// TwinCAT 3 PLC project PLC_Main
// ProgramVersion: 3.1.4026.13
// CompilerDefines: VISU_USEWSTRING
// libraries:
//   Tc2_Standard, * (Beckhoff Automation GmbH)
//   Tc2_System, * (Beckhoff Automation GmbH)
//   Tc3_Module, * (Beckhoff Automation GmbH)
// project tree:
//   DUTs/ DUT_TestStruct.TcDUT, DUT_TestStruct2.TcDUT, MonitorTest.TcDUT, MonitorTestData.TcDUT, ReadTest.TcDUT, ReadTestData.TcDUT, SymbolTest.TcDUT, TestEnum.TcDUT, WriteTest.TcDUT, WriteTestData.TcDUT
//   GVLs/ AdsNet8.TcGVL, AdsNet9.TcGVL, OpcNet8.TcGVL, OpcNet9.TcGVL
//   / PlcTask.TcTTO
//   POUs/ MAIN.TcPOU, ResetWriteData.TcPOU
// real-time tasks:
//   TASK PlcTask: cycle T#10ms, priority 20, ADS port 350

CONFIGURATION PLC_Main
    RESOURCE PLC ON TwinCAT3
        TASK PlcTask(INTERVAL := T#10ms, PRIORITY := 20);
        PROGRAM MAIN WITH PlcTask : MAIN;
    END_RESOURCE
END_CONFIGURATION

// ---- DUTs/DUT_TestStruct.TcDUT
{attribute 'analysis' := '-33'}
TYPE DUT_TestStruct :
STRUCT
	BoolValue						:BOOL			:= TRUE;
	
	ByteValue						:BYTE			:= 16#FF;
	WordValue						:WORD			:= 16#FFFF;
	DWordValue						:DWORD			:= 16#FFFF_FFFF;
	LWordValue						:LWORD			:= 16#FFFF_FFFF_FFFF_FFFF;
	
	ShortValue						:SINT			:= -128;
	IntValue						:INT			:= -32768;
	DIntValue						:DINT			:= -2147483648 ;
	LongValue						:LINT			:= -9223372036854775808;

	UShortValue						:USINT			:= 255;
	UIntValue						:UINT			:= 65535;
	UDIntValue						:UDINT			:= 4294967295;
	ULongValue						:ULINT			:= 18446744073709551615;
										   
	FloatValue						:REAL			:= -3.402823E+38;
	DoubleValue						:LREAL			:= -1.79769313486231E+308;
	
	TimeValue						:TIME			:= T#1000MS;
	TimeOfDay						:TIME_OF_DAY	:= TOD#01:00;
	LTimeValue						:LTIME 			:= LTIME#1000NS;
	DateValue						:DATE			:= D#2106-02-05;
	DateAndTimeValue				:DATE_AND_TIME	:= DT#2106-02-05-06:28:15;
	
	StringValue						:STRING			:= 'Test String';
	WStringValue					:WSTRING		:= "Test WString";
	
	Nested							:DUT_TestStruct2;
	
	IntArray						:ARRAY[0..10] OF INT := [1000, 1001, 1002, 1003, 1004, 1005, 1006, 1007, 1008, 1009, 1010];
	MultiDimensionArray 			:ARRAY[0..1,0..2,0..3] OF INT := [100, 200, 300, 400, 500, 600, 700, 800, 900, 1000, 1100, 1200, 1300, 1400, 1500, 1600, 1700, 1800, 1900, 2000, 2100, 2200, 2300, 2400];
	ComplexArray					:ARRAY[0..2] OF DUT_TestStruct2;
	MultiDimensionComplexArray 		:ARRAY[0..1,0..2,0..3] OF DUT_TestStruct2;
	
	IntArray2						:ARRAY[1..11] OF INT := [1000, 1001, 1002, 1003, 1004, 1005, 1006, 1007, 1008, 1009, 1010];
	MultiDimensionArray2			:ARRAY[1..2,1..3,1..4] OF INT := [100, 200, 300, 400, 500, 600, 700, 800, 900, 1000, 1100, 1200, 1300, 1400, 1500, 1600, 1700, 1800, 1900, 2000, 2100, 2200, 2300, 2400];
	ComplexArray2					:ARRAY[1..3] OF DUT_TestStruct2;
	MultiDimensionComplexArray2		:ARRAY[1..2,1..3,1..4] OF DUT_TestStruct2;
END_STRUCT
END_TYPE

// ---- DUTs/DUT_TestStruct2.TcDUT
{attribute 'analysis' := '-33'}
TYPE DUT_TestStruct2 :
STRUCT
	ByteValue			:BYTE			:= 16#FF;
	WordValue			:WORD			:= 16#FFFF;
	DWordValue			:DWORD			:= 16#FFFF_FFFF;
	LWordValue			:LWORD			:= 16#FFFF_FFFF_FFFF_FFFF;
END_STRUCT
END_TYPE

// ---- DUTs/MonitorTest.TcDUT
{attribute 'analysis' := '-33'}
TYPE MonitorTest :
STRUCT
    MonitorBeforeConnectDoesNotMatter			: BOOL;	
    SubscriptionsWillAllTriggerOnUpdateAsync	: BOOL;
    RegisterUnregisterIO						: BOOL;
    
    RegisterUnregisterMultipleIO1				: BOOL;
    RegisterUnregisterMultipleIO2				: BOOL;
    RegisterUnregisterMultipleIO3				: BOOL;
    RegisterUnregisterMultipleIO4				: BOOL;
    RegisterUnregisterMultipleIO5				: BOOL;
    RegisterUnregisterMultipleIO6				: BOOL;
    RegisterUnregisterMultipleIO7				: BOOL;
    RegisterUnregisterMultipleIO8				: BOOL;
    
    SubscribeIOUpdatesWhenValueChanges			: BOOL;
    SubscriptionsPersistReconnects				: BOOL;
    SubscribeIOShouldTriggerOnSubscribe			: BOOL;
    
    CanSubscribeToAllPlcTypes					: MonitorTestData;
END_STRUCT
END_TYPE

// ---- DUTs/MonitorTestData.TcDUT
{attribute 'analysis' := '-33'}
TYPE MonitorTestData :
STRUCT
	BoolValue			: BOOL;
	
	ByteValue			: BYTE;
	WordValue			: WORD;
	DWordValue			: DWORD;
	LWordValue			: LWORD;
	
	SIntValue			: SINT;
	IntValue			: INT;
	DIntValue			: DINT;
	LIntValue			: LINT;
	
	USIntValue			: USINT;
	UIntValue			: UINT;
	UDIntValue			: UDINT;
	ULIntValue			: ULINT;
	
	RealValue			: REAL;
	LRealValue			: LREAL;
	
	TimeValue			: TIME;
	TimeOfDayValue		: TOD;
	LTimeValue			: LTIME;
	DateValue			: DATE;
	DateAndTimeValue	: DT;
	StringValue			: STRING;
	WStringValue		: WSTRING;
	EnumValue1			: TestEnum;
	EnumValue2			: TestEnum;
END_STRUCT
END_TYPE

// ---- DUTs/ReadTest.TcDUT
{attribute 'analysis' := '-33'}
TYPE ReadTest :
STRUCT
	ReadDynamicReadsAStructure					: DUT_TestStruct;
	ReadDynamicReadsAStructureAsync				: DUT_TestStruct;

	ReadGenericReturnsTheRequestedType			: ReadTestData;
	ReadGenericReturnsTheRequestedTypeAsync		: ReadTestData;
	
	ReadMultipleItemsInOneTransaction			: ReadTestData;
	ReadMultipleItemsInOneTransactionAsync		: ReadTestData;
	
	ReadValueReturnsTheExpectedValue			: ReadTestData;
	ReadValueReturnsTheExpectedValueAsync		: ReadTestData;
	
	WaitForValueThrowsExceptionOnTimeout		: BOOL;
	WaitForValueThrowsExceptionOnTimeoutAsync	: BOOL;
	
	WaitsForValueToChange						: ReadTestData;
	WaitsForValueToChangeAsync					: ReadTestData;
END_STRUCT
END_TYPE

// ---- DUTs/ReadTestData.TcDUT
{attribute 'analysis' := '-33'}
TYPE ReadTestData :
STRUCT
	BoolValue						: BOOL := TRUE;
	ByteValue						: BYTE := 16#FF;
	WordValue						: WORD := 16#FFFF;
	DWordValue						: DWORD := 16#FFFF_FFFF;
	LWordValue						: LWORD := 16#FFFF_FFFF_FFFF_FFFF;
	SIntValue						: SINT := -128;
	IntValue						: INT := -32768;
	DIntValue						: DINT := -2147483648;
	LIntValue						: LINT := -9223372036854775808;
	USIntValue						: USINT := 255;
	UIntValue						: UINT := 65535;
	UDIntValue						: UDINT := 4294967295;
	ULIntValue						: ULINT := 18446744073709551615;
	RealValue						: REAL := -3.402823E+38;
	LRealValue						: LREAL := -1.79769313486231E+308;
	TimeValue						: TIME := T#1000MS;
	TimeOfDayValue					: TOD := TOD#01:00;
	LTimeValue						: LTIME := LTIME#1000NS;
	DateValue						: DATE := D#2106-02-05;
	DateAndTimeValue				: DT := DT#2106-02-05-06:28:15;
	StringValue						: STRING := 'Test String';
	WStringValue					: WSTRING := "Test WString";
	EnumValue1						: TestEnum := TestEnum.second;
	EnumValue2						: TestEnum := TestEnum.second;
	
	IntArray						: ARRAY[0..10] OF INT := [1000, 1001, 1002, 1003, 1004, 1005, 1006, 1007, 1008, 1009, 1010];
	MultiDimensionArray 			: ARRAY[0..1,0..2,0..3] OF INT := [100, 200, 300, 400, 500, 600, 700, 800, 900, 1000, 1100, 1200, 1300, 1400, 1500, 1600, 1700, 1800, 1900, 2000, 2100, 2200, 2300, 2400];
	ComplexArray					: ARRAY[0..2] OF DUT_TestStruct2;
	MultiDimensionComplexArray 		: ARRAY[0..1,0..2,0..3] OF DUT_TestStruct2;
	
	IntArray2						: ARRAY[1..11] OF INT := [1000, 1001, 1002, 1003, 1004, 1005, 1006, 1007, 1008, 1009, 1010];
	MultiDimensionArray2 			: ARRAY[1..2,1..3,1..4] OF INT := [100, 200, 300, 400, 500, 600, 700, 800, 900, 1000, 1100, 1200, 1300, 1400, 1500, 1600, 1700, 1800, 1900, 2000, 2100, 2200, 2300, 2400];
	ComplexArray2					: ARRAY[1..3] OF DUT_TestStruct2;
	MultiDimensionComplexArray2		: ARRAY[1..2,1..3,1..4] OF DUT_TestStruct2;
	
	StructValue						: DUT_TestStruct;
	StructValue2					: DUT_TestStruct;
END_STRUCT
END_TYPE

// ---- DUTs/SymbolTest.TcDUT
{attribute 'analysis' := '-33'}
TYPE SymbolTest :
STRUCT
	GetSymbolInfoReturnsTheSymbol				: BOOL;
	TryGetSymbolInfoReturnsTrueWithValidData	: BOOL;
END_STRUCT
END_TYPE

// ---- DUTs/TestEnum.TcDUT
{attribute 'qualified_only'}
{attribute 'strict'}
TYPE TestEnum :
(
	first := 0,
	second := 1,
	third := 2
);
END_TYPE

// ---- DUTs/WriteTest.TcDUT
TYPE WriteTest :
STRUCT
	ToggleBool								: BOOL;
	
	WriteGenericUpdatesTheValueInPlc		: WriteTestData;
	WriteGenericUpdatesTheValueInPlcAsync	: WriteTestData;
	
	WriteMultipleUpdatesTheValueInPlc		: WriteTestData;
	WriteMultipleUpdatesTheValueInPlcAsync	: WriteTestData;
	
	WriteUpdatesTheValueInPlc				: WriteTestData;
	WriteUpdatesTheValueInPlcAsync			: WriteTestData;
END_STRUCT
END_TYPE

// ---- DUTs/WriteTestData.TcDUT
TYPE WriteTestData :
STRUCT
	Reset								: BOOL 			:= FALSE;
	
	BoolValueReset						: BOOL			:= FALSE;
	BoolValue							: BOOL			:= TRUE;
	
	ByteValueReset						: BOOL			:= FALSE;
	ByteValue							: BYTE			:= 16#FF;
	WordValueReset						: BOOL			:= FALSE;
	WordValue							: WORD			:= 16#FFFF;
	DWordValueReset						: BOOL			:= FALSE;
	DWordValue							: DWORD			:= 16#FFFF_FFFF;
	LWordValueReset						: BOOL			:= FALSE;
	LWordValue							: LWORD			:= 16#FFFF_FFFF_FFFF_FFFF;
	
	SIntValueReset						: BOOL			:= FALSE;
	SIntValue							: SINT			:= -128;
	IntValueReset						: BOOL			:= FALSE;
	IntValue							: INT			:= -32768;
	DIntValueReset						: BOOL			:= FALSE;
	DIntValue							: DINT			:= -2147483648 ;
	LIntValueReset						: BOOL			:= FALSE;
	LIntValue							: LINT			:= -9223372036854775808;
	
	USIntValueReset						: BOOL			:= FALSE;
	USIntValue							: USINT			:= 255;
	UIntValueReset						: BOOL			:= FALSE;
	UIntValue							: UINT			:= 65535;
	UDIntValueReset						: BOOL			:= FALSE;
	UDIntValue							: UDINT			:= 4294967295;
	ULIntValueReset						: BOOL			:= FALSE;
	ULIntValue							: ULINT			:= 18446744073709551615;
	
	RealValueReset						: BOOL			:= FALSE;
	RealValue							: REAL			:= -3.402823E+38;
	LRealValueReset						: BOOL			:= FALSE;
	LRealValue							: LREAL			:= -1.79769313486231E+308;
	
	TimeValue1Reset						: BOOL			:= FALSE;
	TimeValue1							: TIME			:= T#1000MS;
	TimeValue2Reset						: BOOL			:= FALSE;
	TimeValue2							: TIME			:= T#1000MS;
	TimeOfDayValue1Reset				: BOOL			:= FALSE;
	TimeOfDayValue1						: TIME_OF_DAY	:= TOD#01:00;
	TimeOfDayValue2Reset				: BOOL			:= FALSE;
	TimeOfDayValue2						: TIME_OF_DAY	:= TOD#01:00;
	LTimeValue1Reset					: BOOL			:= FALSE;
	LTimeValue1							: LTIME 		:= LTIME#1000NS;
	LTimeValue2Reset					: BOOL			:= FALSE;
	LTimeValue2							: LTIME 		:= LTIME#1000NS;
	DateValue1Reset						: BOOL			:= FALSE;
	DateValue1							: DATE			:= D#2106-02-06;
	DateValue2Reset						: BOOL			:= FALSE;
	DateValue2							: DATE			:= D#2106-02-06;
	DateAndTimeValue1Reset				: BOOL			:= FALSE;
	DateAndTimeValue1					: DATE_AND_TIME	:= DT#2106-02-06-06:28:15;
	DateAndTimeValue2Reset				: BOOL			:= FALSE;
	DateAndTimeValue2					: DATE_AND_TIME	:= DT#2106-02-06-06:28:15;
	
	StringValueReset					: BOOL			:= FALSE;
	StringValue							: STRING		:= 'Test String';
	WStringValueReset					: BOOL			:= FALSE;
	WStringValue						: WSTRING		:= "Test WString";
	
	EnumValue1Reset						: BOOL			:= FALSE;
	EnumValue1							: TestEnum		:= TestEnum.first;
	EnumValue2Reset						: BOOL			:= FALSE;
	EnumValue2							: TestEnum		:= TestEnum.first;
	EnumValue3Reset						: BOOL			:= FALSE;
	EnumValue3							: TestEnum		:= TestEnum.first;
	
	IntArrayReset						: BOOL			:= FALSE;
	IntArray							: ARRAY[0..10] OF INT := [1000, 1001, 1002, 1003, 1004, 1005, 1006, 1007, 1008, 1009, 1010];
	MultiDimensionArrayReset			: BOOL			:= FALSE;
	MultiDimensionArray 				: ARRAY[0..1,0..2,0..3] OF INT := [100, 200, 300, 400, 500, 600, 700, 800, 900, 1000, 1100, 1200, 1300, 1400, 1500, 1600, 1700, 1800, 1900, 2000, 2100, 2200, 2300, 2400];
	ComplexArrayReset					: BOOL			:= FALSE;
	ComplexArray						: ARRAY[0..2] OF DUT_TestStruct2;
	MultiDimensionComplexArrayReset		: BOOL			:= FALSE;
	MultiDimensionComplexArray 			: ARRAY[0..1,0..2,0..3] OF DUT_TestStruct2;
	
	IntArray2Reset						: BOOL			:= FALSE;
	IntArray2							: ARRAY[1..11] OF INT := [1000, 1001, 1002, 1003, 1004, 1005, 1006, 1007, 1008, 1009, 1010];
	MultiDimensionArray2Reset			: BOOL			:= FALSE;
	MultiDimensionArray2 				: ARRAY[1..2,1..3,1..4] OF INT := [100, 200, 300, 400, 500, 600, 700, 800, 900, 1000, 1100, 1200, 1300, 1400, 1500, 1600, 1700, 1800, 1900, 2000, 2100, 2200, 2300, 2400];
	ComplexArray2Reset					: BOOL			:= FALSE;
	ComplexArray2						: ARRAY[1..3] OF DUT_TestStruct2;
	MultiDimensionComplexArray2Reset	: BOOL			:= FALSE;
	MultiDimensionComplexArray2 		: ARRAY[1..2,1..3,1..4] OF DUT_TestStruct2;
	
	Nested1Reset						: BOOL			:= FALSE;
	Nested1								: DUT_TestStruct2;
	Nested2Reset						: BOOL			:= FALSE;
	Nested2								: DUT_TestStruct2;
	
	StructValue1Reset					: BOOL			:= FALSE;
	StructValue1						: DUT_TestStruct;
	StructValue2Reset					: BOOL			:= FALSE;
	StructValue2						: DUT_TestStruct;
END_STRUCT
END_TYPE

// ---- GVLs/AdsNet8.TcGVL
{attribute 'qualified_only'}
{attribute 'analysis' := '-33'}
VAR_GLOBAL
	MonitorTestData		: MonitorTest;
	ReadTestData		: ReadTest;
	SymbolTestData		: SymbolTest;
	WriteTestData		: WriteTest;
END_VAR

// ---- GVLs/AdsNet9.TcGVL
{attribute 'qualified_only'}
{attribute 'analysis' := '-33'}
VAR_GLOBAL
	MonitorTestData		: MonitorTest;
	ReadTestData		: ReadTest;
	SymbolTestData		: SymbolTest;
	WriteTestData		: WriteTest;
END_VAR

// ---- GVLs/OpcNet8.TcGVL
{attribute 'qualified_only'}
{attribute 'analysis' := '-33'}
VAR_GLOBAL
	{attribute 'OPC.UA.DA' := '1'}
	MonitorTestData		: MonitorTest;
	{attribute 'OPC.UA.DA' := '1'}
	ReadTestData		: ReadTest;
	{attribute 'OPC.UA.DA' := '1'}
	SymbolTestData		: SymbolTest;
	{attribute 'OPC.UA.DA' := '1'}
	WriteTestData		: WriteTest;
END_VAR

// ---- GVLs/OpcNet9.TcGVL
{attribute 'qualified_only'}
{attribute 'analysis' := '-33'}
VAR_GLOBAL
	{attribute 'OPC.UA.DA' := '1'}
	MonitorTestData		: MonitorTest;
	{attribute 'OPC.UA.DA' := '1'}
	ReadTestData		: ReadTest;
	{attribute 'OPC.UA.DA' := '1'}
	SymbolTestData		: SymbolTest;
	{attribute 'OPC.UA.DA' := '1'}
	WriteTestData		: WriteTest;
END_VAR

// ---- POUs/MAIN.TcPOU
PROGRAM MAIN

ResetWriteData(AdsNet8.WriteTestData.WriteGenericUpdatesTheValueInPlc);
ResetWriteData(AdsNet8.WriteTestData.WriteGenericUpdatesTheValueInPlcAsync);
ResetWriteData(AdsNet8.WriteTestData.WriteMultipleUpdatesTheValueInPlc);
ResetWriteData(AdsNet8.WriteTestData.WriteMultipleUpdatesTheValueInPlcAsync);
ResetWriteData(AdsNet8.WriteTestData.WriteUpdatesTheValueInPlc);
ResetWriteData(AdsNet8.WriteTestData.WriteUpdatesTheValueInPlcAsync);

ResetWriteData(AdsNet9.WriteTestData.WriteGenericUpdatesTheValueInPlc);
ResetWriteData(AdsNet9.WriteTestData.WriteGenericUpdatesTheValueInPlcAsync);
ResetWriteData(AdsNet9.WriteTestData.WriteMultipleUpdatesTheValueInPlc);
ResetWriteData(AdsNet9.WriteTestData.WriteMultipleUpdatesTheValueInPlcAsync);
ResetWriteData(AdsNet9.WriteTestData.WriteUpdatesTheValueInPlc);
ResetWriteData(AdsNet9.WriteTestData.WriteUpdatesTheValueInPlcAsync);

ResetWriteData(OpcNet8.WriteTestData.WriteGenericUpdatesTheValueInPlc);
ResetWriteData(OpcNet8.WriteTestData.WriteGenericUpdatesTheValueInPlcAsync);
ResetWriteData(OpcNet8.WriteTestData.WriteMultipleUpdatesTheValueInPlc);
ResetWriteData(OpcNet8.WriteTestData.WriteMultipleUpdatesTheValueInPlcAsync);
ResetWriteData(OpcNet8.WriteTestData.WriteUpdatesTheValueInPlc);
ResetWriteData(OpcNet8.WriteTestData.WriteUpdatesTheValueInPlcAsync);

ResetWriteData(OpcNet9.WriteTestData.WriteGenericUpdatesTheValueInPlc);
ResetWriteData(OpcNet9.WriteTestData.WriteGenericUpdatesTheValueInPlcAsync);
ResetWriteData(OpcNet9.WriteTestData.WriteMultipleUpdatesTheValueInPlc);
ResetWriteData(OpcNet9.WriteTestData.WriteMultipleUpdatesTheValueInPlcAsync);
ResetWriteData(OpcNet9.WriteTestData.WriteUpdatesTheValueInPlc);
ResetWriteData(OpcNet9.WriteTestData.WriteUpdatesTheValueInPlcAsync);

END_PROGRAM

// ---- POUs/ResetWriteData.TcPOU
FUNCTION ResetWriteData : BOOL
VAR_INPUT
	data			: REFERENCE TO WriteTestData;
END_VAR
VAR CONSTANT
	EmptyStruct		: DUT_TestStruct;
END_VAR

IF data.Reset THEN
	data.BoolValue						:= TRUE;
	
	data.ByteValue						:= 16#FF;
	data.WordValue						:= 16#FFFF;
	data.DWordValue						:= 16#FFFF_FFFF;
	data.LWordValue						:= 16#FFFF_FFFF_FFFF_FFFF;

	data.SIntValue						:= -128;
	data.IntValue						:= -32768;
	data.DIntValue						:= -2147483648 ;
	data.LIntValue						:= -9223372036854775808;

	data.USIntValue						:= 255;
	data.UIntValue						:= 65535;
	data.UDIntValue						:= 4294967295;
	data.ULintValue						:= 18446744073709551615;
	
	data.RealValue						:= -3.402823E+38;
	data.LRealValue						:= -1.79769313486231E+308;
	
	data.TimeValue1						:= T#1000MS;
	data.TimeValue2						:= T#1000MS;
	data.TimeOfDayValue1				:= TOD#01:00;
	data.TimeOfDayValue2				:= TOD#01:00;
	data.LTimeValue1					:= LTIME#1000NS;
	data.LTimeValue2					:= LTIME#1000NS;
	data.DateValue1						:= D#2106-02-06;
	data.DateValue2						:= D#2106-02-06;
	data.DateAndTimeValue1				:= DT#2106-02-06-06:28:15;
	data.DateAndTimeValue2				:= DT#2106-02-06-06:28:15;
	
	data.StringValue					:= 'Test String';
	data.WStringValue					:= "Test WString";
	
	data.EnumValue1						:= TestEnum.first;
	data.EnumValue2						:= TestEnum.first;
	data.EnumValue3						:= TestEnum.first;
	
	data.IntArray				 		:= EmptyStruct.IntArray;	
	data.MultiDimensionArray			:= EmptyStruct.MultiDimensionArray;
	data.ComplexArray					:= EmptyStruct.ComplexArray;
	data.MultiDimensionComplexArray		:= EmptyStruct.MultiDimensionComplexArray;
	
	data.IntArray2				 		:= EmptyStruct.IntArray2;	
	data.MultiDimensionArray2			:= EmptyStruct.MultiDimensionArray2;
	data.ComplexArray2					:= EmptyStruct.ComplexArray2;
	data.MultiDimensionComplexArray2	:= EmptyStruct.MultiDimensionComplexArray2;
	
	data.Nested1						:= EmptyStruct.Nested;
	data.Nested2						:= EmptyStruct.Nested;
	data.StructValue1					:= EmptyStruct;
	data.StructValue2					:= EmptyStruct;
	
	data.Reset 							:= FALSE;
END_IF

IF (data.BoolValueReset) THEN
	data.BoolValue						:= TRUE;
	data.BoolValueReset					:= FALSE;
END_IF
	
IF (data.ByteValueReset) THEN
	data.ByteValue						:= 16#FF;
	data.ByteValueReset					:= FALSE;
END_IF
	
IF (data.WordValueReset) THEN
	data.WordValue						:= 16#FFFF;
	data.WordValueReset					:= FALSE;
END_IF
	
IF (data.DWordValueReset) THEN
	data.DWordValue						:= 16#FFFF_FFFF;
	data.DWordValueReset				:= FALSE;
END_IF
	
IF (data.LWordValueReset) THEN
	data.LWordValue						:= 16#FFFF_FFFF_FFFF_FFFF;
	data.LWordValueReset				:= FALSE;
END_IF
	
IF (data.SIntValueReset) THEN
	data.SIntValue						:= -128;
	data.SIntValueReset					:= FALSE;
END_IF
	
IF (data.IntValueReset) THEN
	data.IntValue						:= -32768;
	data.IntValueReset					:= FALSE;
END_IF
	
IF (data.DIntValueReset) THEN
	data.DIntValue						:= -2147483648 ;
	data.DIntValueReset					:= FALSE;
END_IF
	
IF (data.LIntValueReset) THEN
	data.LIntValue						:= -9223372036854775808;
	data.LIntValueReset					:= FALSE;
END_IF
	
IF (data.USIntValueReset) THEN
	data.USIntValue						:= 255;
	data.USIntValueReset				:= FALSE;
END_IF
	
IF (data.UIntValueReset) THEN
	data.UIntValue						:= 65535;
	data.UIntValueReset					:= FALSE;
END_IF
	
IF (data.UDIntValueReset) THEN
	data.UDIntValue						:= 4294967295;
	data.UDIntValueReset				:= FALSE;
END_IF
	
IF (data.ULintValueReset) THEN
	data.ULintValue						:= 18446744073709551615;
	data.ULintValueReset					:= FALSE;
END_IF
	
IF (data.RealValueReset) THEN
	data.RealValue						:= -3.402823E+38;
	data.RealValueReset					:= FALSE;
END_IF
	
IF (data.LRealValueReset) THEN
	data.LRealValue						:= -1.79769313486231E+308;
	data.LRealValueReset				:= FALSE;
END_IF
	
IF (data.TimeValue1Reset) THEN
	data.TimeValue1						:= T#1000MS;
	data.TimeValue1Reset				:= FALSE;
END_IF
	
IF (data.TimeValue2Reset) THEN
	data.TimeValue2						:= T#1000MS;
	data.TimeValue2Reset				:= FALSE;
END_IF
	
IF (data.TimeOfDayValue1Reset) THEN
	data.TimeOfDayValue1				:= TOD#01:00;
	data.TimeOfDayValue1Reset			:= FALSE;
END_IF
	
IF (data.TimeOfDayValue2Reset) THEN
	data.TimeOfDayValue2				:= TOD#01:00;
	data.TimeOfDayValue2Reset			:= FALSE;
END_IF
	
IF (data.LTimeValue1Reset) THEN
	data.LTimeValue1					:= LTIME#1000NS;
	data.LTimeValue1Reset				:= FALSE;
END_IF
	
IF (data.LTimeValue2Reset) THEN
	data.LTimeValue2					:= LTIME#1000NS;
	data.LTimeValue2Reset				:= FALSE;
END_IF
	
IF (data.DateValue1Reset) THEN
	data.DateValue1						:= D#2106-02-06;
	data.DateValue1Reset				:= FALSE;
END_IF
	
IF (data.DateValue2Reset) THEN
	data.DateValue2						:= D#2106-02-06;
	data.DateValue2Reset				:= FALSE;
END_IF
	
IF (data.DateAndTimeValue1Reset) THEN
	data.DateAndTimeValue1				:= DT#2106-02-06-06:28:15;
	data.DateAndTimeValue1Reset			:= FALSE;
END_IF
	
IF (data.DateAndTimeValue2Reset) THEN
	data.DateAndTimeValue2				:= DT#2106-02-06-06:28:15;
	data.DateAndTimeValue2Reset			:= FALSE;
END_IF
	
IF (data.StringValueReset) THEN
	data.StringValue					:= 'Test String';
	data.StringValueReset				:= FALSE;
END_IF
	
IF (data.WStringValueReset) THEN
	data.WStringValue					:= "Test WString";
	data.WStringValueReset				:= FALSE;
END_IF
	
IF (data.EnumValue1Reset) THEN
	data.EnumValue1						:= TestEnum.first;
	data.EnumValue1Reset				:= FALSE;
END_IF
	
IF (data.EnumValue2Reset) THEN
	data.EnumValue2						:= TestEnum.first;
	data.EnumValue2Reset				:= FALSE;
END_IF
	
IF (data.EnumValue3Reset) THEN
	data.EnumValue3						:= TestEnum.first;
	data.EnumValue3Reset				:= FALSE;
END_IF
	
IF (data.IntArrayReset) THEN
	data.IntArray				 		:= EmptyStruct.IntArray;
	data.IntArrayReset					:= FALSE;
END_IF
	
IF (data.MultiDimensionArrayReset) THEN
	data.MultiDimensionArray			:= EmptyStruct.MultiDimensionArray;
	data.MultiDimensionArrayReset		:= FALSE;
END_IF
	
IF (data.ComplexArrayReset) THEN
	data.ComplexArray					:= EmptyStruct.ComplexArray;
	data.ComplexArrayReset				:= FALSE;
END_IF
	
IF (data.MultiDimensionComplexArrayReset) THEN
	data.MultiDimensionComplexArray		:= EmptyStruct.MultiDimensionComplexArray;
	data.MultiDimensionComplexArrayReset:= FALSE;
END_IF

IF (data.IntArray2Reset) THEN
	data.IntArray2				 		:= EmptyStruct.IntArray2;
	data.IntArray2Reset					:= FALSE;
END_IF
	
IF (data.MultiDimensionArray2Reset) THEN
	data.MultiDimensionArray2			:= EmptyStruct.MultiDimensionArray2;
	data.MultiDimensionArray2Reset		:= FALSE;
END_IF
	
IF (data.ComplexArray2Reset) THEN
	data.ComplexArray2					:= EmptyStruct.ComplexArray2;
	data.ComplexArray2Reset				:= FALSE;
END_IF
	
IF (data.MultiDimensionComplexArray2Reset) THEN
	data.MultiDimensionComplexArray2		:= EmptyStruct.MultiDimensionComplexArray2;
	data.MultiDimensionComplexArray2Reset:= FALSE;
END_IF
	
IF (data.Nested1Reset) THEN
	data.Nested1						:= EmptyStruct.Nested;
	data.Nested1Reset:= FALSE;
END_IF
	
IF (data.Nested2Reset) THEN
	data.Nested2						:= EmptyStruct.Nested;
	data.Nested2Reset:= FALSE;
END_IF
	
IF (data.StructValue1Reset) THEN
	data.StructValue1					:= EmptyStruct;
	data.StructValue1Reset:= FALSE;
END_IF
	
IF (data.StructValue2Reset) THEN
	data.StructValue2					:= EmptyStruct;
	data.StructValue2Reset:= FALSE;
END_IF

END_FUNCTION
